PROGRAM PRG_ThreeDOF_robot_TEST
VAR
END_VAR

END_PROGRAM

(* stored: Version 1.1.0.1, ProductVersion 3.1.4024.13
   POU PRG_ThreeDOF_robot_TEST: Id {e4d7c900-4ddd-4d6a-8b55-ef2e1fbec25d}, SpecialFunc None *)
